PROGRAM P_ReadCsv
VAR
END_VAR

END_PROGRAM

(* stored: Version 1.1.0.1, ProductVersion 3.1.4024.3
   POU P_ReadCsv: Id {c07ebfae-1465-4e3d-97c4-9ee68704ec42}, SpecialFunc None *)
